// TIA Portal V20 export
// export: Created 2026-07-23T04:47:09.98054Z, ExportSetting WithDefaults, DisplayName Totally Integrated Automation Portal, DisplayVersion V20, DisplayName TIA Portal Openness, DisplayVersion V20, DisplayName TIA Portal Version Control Interface, DisplayVersion V20, DisplayName STEP 7 Professional, DisplayVersion V20, DisplayName STEP 7 Safety, DisplayVersion V20, DisplayName WinCC Basic/Comfort/Advanced, DisplayVersion V20, DisplayName WinCC Professional, DisplayVersion V20, DisplayName WinCC Unified, DisplayVersion V20
LibraryTypeVersion   Author=TIA_VM, VersionNumber=0.0.1
